ABB RobotStudio station: kabil box moving.rsstn

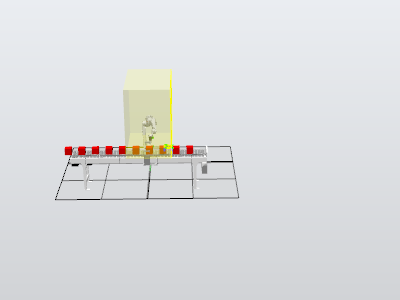
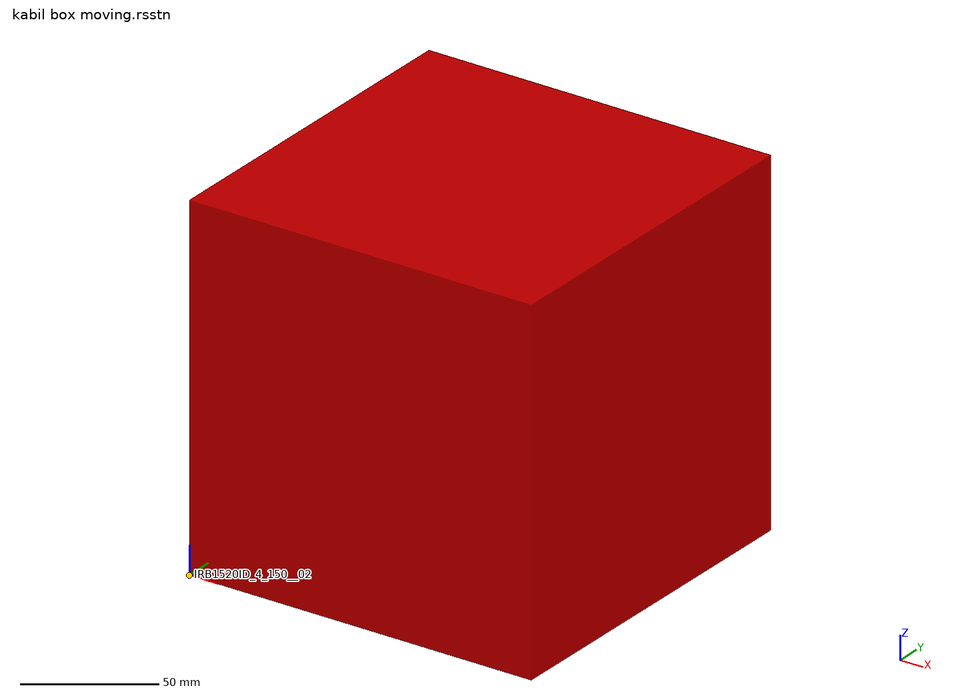
[picture v1: parts stored in the station drawn from their meshes, with robot base, taught points and paths (robot models come from the ABB library and are not in the file)]
Station Station (saved by RobotStudio 22.3.10141.1)
Controller Controller13, task T_ROB1: task frame (RAPID world) sits at (-531.75, 1087.38, 775) mm in the station
Controller Controller13
  mechanical unit ROB_1: IRB1520ID_4_150__02, 6 joints, base frame (531.75, -1087.38, -775) mm, rotated rx 0 ry 0 rz 90 deg
  mechanical unit CNV1: ?, 1 joints, base frame (0, 0, 0) mm
Layout (positions relative to the parent item):
  - IRB1520ID_4_150__02 [mechanism, from Robots\IRB1520ID_4_150_G_02.rslib] at (0, 0, 0) mm, rotated rx 0 ry 0 rz 90 deg; joint values [0.0771, -0.2955, 0.4507, -0.183, 0.3754, 0.2092] (rad or m)
  - MyTool [mechanism, from Training Objects\myTool.rslib] at (-56.52, 904.41, 1003.29) mm, rotated rx -180 ry 60 rz -90 deg
  - Conveyor [conveyor]
    - 400_guide [part] at (-1306.59, 1084.88, 0) mm, size 3033 x 590 x 945 mm
    - Part_1 [part], size 150 x 150 x 150 mm
    - ConveyorObject_98 [conveyorobject] at (1684.25, 1087.38, 775) mm
      - Part_1 [part] at (0, 100, 0) mm, size 150 x 150 x 150 mm
    - ConveyorObject_99 [conveyorobject] at (1384.25, 1087.38, 775) mm
      - Part_1 [part] at (0, 100, 0) mm, size 150 x 150 x 150 mm
    - ConveyorObject_100 [conveyorobject] at (1084.25, 1087.38, 775) mm
      - Part_1 [part] at (0, 100, 0) mm, size 150 x 150 x 150 mm
    - ConveyorObject_101 [conveyorobject] at (784.25, 1087.38, 775) mm
      - Part_1 [part] at (0, 100, 0) mm, size 150 x 150 x 150 mm
    - ConveyorObject_102 [conveyorobject] at (484.25, 1087.38, 775) mm
      - Part_1 [part] at (0, 100, 0) mm, size 150 x 150 x 150 mm
    - ConveyorObject_103 [conveyorobject] at (184.25, 1087.38, 775) mm
      - Part_1 [part] at (0, 100, 0) mm, size 150 x 150 x 150 mm
    - ConveyorObject_104 [conveyorobject] at (-115.75, 1087.38, 775) mm
      - Part_1 [part] at (0, 100, 0) mm, size 150 x 150 x 150 mm
    - ConveyorObject_105 [conveyorobject] at (-415.75, 1087.38, 775) mm
      - Part_1 [part] at (0, 100, 0) mm, size 150 x 150 x 150 mm
    - ConveyorObject_106 [conveyorobject] at (-715.75, 1087.38, 775) mm
      - Part_1 [part] at (0, 100, 0) mm, size 150 x 150 x 150 mm
    - ConveyorObject_107 [conveyorobject] at (-1015.75, 1087.38, 775) mm
      - Part_1 [part] at (0, 100, 0) mm, size 150 x 150 x 150 mm
Attachment: MyTool is attached to IRB1520ID_4_150__02 / Link6
Conveyor tracking Connection_2: unit CNV1, TravelOffset=0.7, QueueTrackDistance=0, StartWindowWidth=1, SyncSeparation=0.1, CountsPerMeter=10000
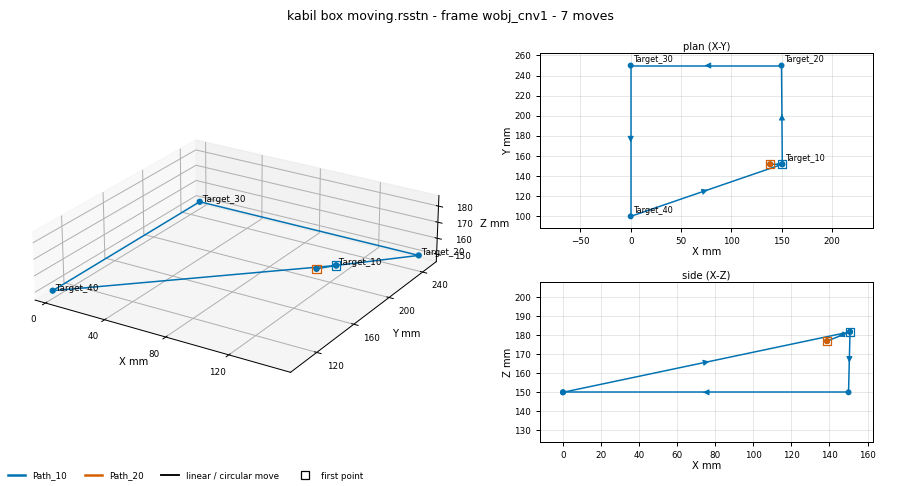
[picture p0: tool path of kabil box moving.rsstn in frame wobj_cnv1, 7 of 7 moves have a stored position in this frame; points joined in program order, loops and branches not executed]
Targets, tools, work objects and paths stored in the station, written as RAPID:
! task T_ROB1
MODULE CalibData
  PERS tooldata MyTool:=[TRUE,[[31.792631019,0,229.638935148],[0.945518576,0,0.325568154,0]],[1,[0,0,1],[1,0,0,0],0,0,0]];
  TASK PERS wobjdata wobj_cnv1:=[FALSE,FALSE,"CNV1",[[0,0,0],[1,0,0,0]],[[0,0,0],[1,0,0,0]]];
ENDMODULE

! task T_ROB1
MODULE Module1
  CONST robtarget home:=[[138.727525622,151.797718786,176.873363016],[0.134922335,-0.694115238,0.694115238,0.134922335],[0,-1,0,0],[9E+09,9E+09,9E+09,9E+09,9E+09,0]];
  CONST robtarget Target_10:=[[150.788156417,151.797837069,181.759926104],[0.134922099,-0.694115318,0.694115255,0.134922073],[0,-1,0,0],[9E+09,9E+09,9E+09,9E+09,9E+09,0]];
  CONST robtarget Target_20:=[[149.999960463,249.999836774,149.999998834],[0.134922026,-0.694115331,0.694115271,0.134921998],[0,-1,0,0],[9E+09,9E+09,9E+09,9E+09,9E+09,0]];
  CONST robtarget Target_30:=[[-0.00003761,249.999827979,149.999976633],[0.13492194,-0.694115341,0.694115291,0.134921926],[0,-1,0,0],[9E+09,9E+09,9E+09,9E+09,9E+09,0]];
  CONST robtarget Target_40:=[[-0.000003009,99.999857704,150.000015395],[0.134921802,-0.694115392,0.694115291,0.134921806],[0,-1,0,0],[9E+09,9E+09,9E+09,9E+09,9E+09,0]];
  PROC Path_10()
    MoveL Target_10,v1000,z100,MyTool\WObj:=wobj_cnv1;
    MoveL Target_20,v1000,z100,MyTool\WObj:=wobj_cnv1;
    MoveL Target_30,v1000,z100,MyTool\WObj:=wobj_cnv1;
    MoveL Target_40,v1000,z100,MyTool\WObj:=wobj_cnv1;
    MoveL Target_10,v1000,z100,MyTool\WObj:=wobj_cnv1;
    MoveL home,v1000,z100,MyTool\WObj:=wobj_cnv1;
  ENDPROC
  PROC Path_20()
    MoveL home,v1000,z100,MyTool\WObj:=wobj_cnv1;
    ActUnit CNV1;
    Path_10;
    WaitWObj wobj_cnv1;
    WaitWObj wobj0;
  ENDPROC
ENDMODULE

